PROGRAM Plc_Prog
VAR
	Motor1 : Motor;
	Motor2 : Motor;
	Motor3 : Motor;
	
	Motor1InputVariables : MotorInputVariables;
	Motor2InputVariables : MotorInputVariables;
	Motor3InputVariables : MotorInputVariables;
	
	Motor1OutputVariables : MotorOutputVariables;
	Motor2OutputVariables : MotorOutputVariables;
	Motor3OutputVariables : MotorOutputVariables;
END_VAR

Motor1(MotorInputs:=Motor1InputVariables, MotorOutputs=>Motor1OutputVariables);
Motor1(MotorInputs:=Motor2InputVariables, MotorOutputs=>Motor2OutputVariables);
Motor1(MotorInputs:=Motor3InputVariables, MotorOutputs=>Motor3OutputVariables);

END_PROGRAM

(* stored: Version 1.1.0.1, ProductVersion 3.1.4024.9
   POU Plc_Prog: Id {ae85b670-d358-4df2-894e-a973366680b5}, SpecialFunc None *)
